(* PLC project PLC, Beckhoff Automation GmbH TwinCAT PLC Control 3.5.13.21 *)
(* stored: creationDateTime 2022-06-22T22:53:30.7833533, modificationDateTime 2022-06-22T22:53:30.7873581 *)

FUNCTION_BLOCK DWORD_TO_BCD
VAR_INPUT
	en: BOOL;
	win: DWORD;
END_VAR
VAR_OUTPUT
	eno: BOOL;
	err: BOOL;
	bout: DWORD;
END_VAR
VAR
	n: DWORD;
	d: DWORD;
	digit: INT;
	base: DWORD;
END_VAR

            err := FALSE;
n := win;
bout := 0;

IF en THEN
	IF win > 99999999 THEN
		err := TRUE;
		RETURN;
	END_IF
	
	FOR digit := 7 TO 0 BY -1 DO
		base := LREAL_TO_DWORD(EXPT(10, digit));
		d := n / base;
		bout := bout + SHL(d, digit * 4);
		n := n - d * base;
	END_FOR
	
	eno := TRUE;
ELSE
	eno := FALSE;
END_IF
          
END_FUNCTION_BLOCK
